SUBAPPLICATION Uebung_006a4 (* SR und T-Flip-Flop mit 3x IE und LinksRechts Baustein *)
  (* Standard: 61499-2; Description: Copyright (c) 2023 Meisterschulen am Ostbahnhof This program and the accompanying materials are made available under the terms of the Eclipse Public License 2.0 which is available at https://www.eclipse.org/legal/epl-2.0/ SPDX-License-Identifier: EPL-2.0 *)
  (* Version 1.0, 2023-10-23, Franz Höpfinger, Meisterschulen am Ostbahnhof *)
  PACKAGE Uebungen;
  IMPORT logiBUS::io::DI::logiBUS_DI::Input_I1;
  IMPORT logiBUS::io::DI::logiBUS_DI::Input_I2;
  IMPORT logiBUS::io::DI::logiBUS_DI::Input_I3;
  IMPORT logiBUS::io::DI::logiBUS_DI_Events::BUTTON_SINGLE_CLICK;
  IMPORT logiBUS::io::DQ::logiBUS_DO::Output_Q1;
  IMPORT logiBUS::io::DQ::logiBUS_DO::Output_Q2;
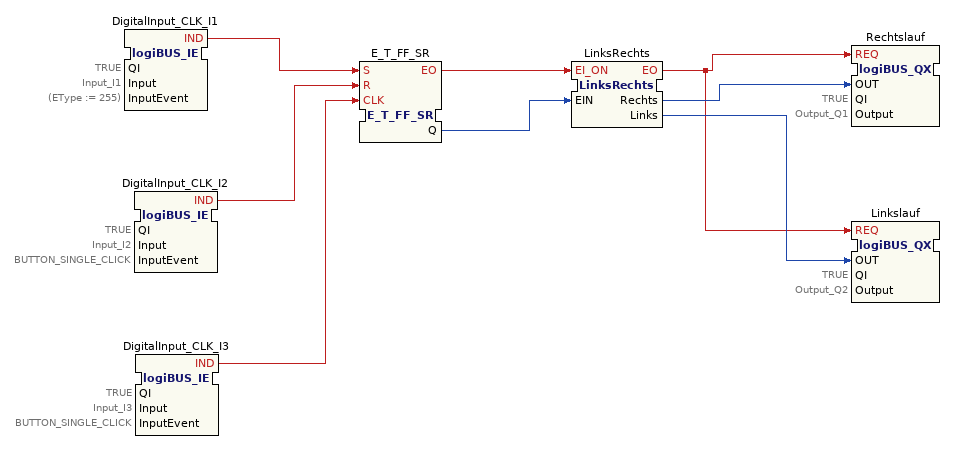
  FBS
    DigitalInput_CLK_I1 : logiBUS::io::DI::logiBUS_IE(QI := TRUE, Input := Input_I1, InputEvent := (EType := 255));
    DigitalInput_CLK_I2 : logiBUS::io::DI::logiBUS_IE(QI := TRUE, Input := Input_I2, InputEvent := BUTTON_SINGLE_CLICK);
    E_T_FF_SR : iec61499::events::E_T_FF_SR;
    DigitalInput_CLK_I3 : logiBUS::io::DI::logiBUS_IE(QI := TRUE, Input := Input_I3, InputEvent := BUTTON_SINGLE_CLICK);
    Rechtslauf : logiBUS::io::DQ::logiBUS_QX(QI := TRUE, Output := Output_Q1);
    Linkslauf : logiBUS::io::DQ::logiBUS_QX(QI := TRUE, Output := Output_Q2);
    LinksRechts : logiBUS::utils::sequence::verteiler::LinksRechts;
  END_FBS
  EVENT_CONNECTIONS
    DigitalInput_CLK_I1.IND TO E_T_FF_SR.S;
    DigitalInput_CLK_I2.IND TO E_T_FF_SR.R;
    DigitalInput_CLK_I3.IND TO E_T_FF_SR.CLK;
    E_T_FF_SR.EO TO LinksRechts.EI_ON;
    LinksRechts.EO TO Linkslauf.REQ;
    LinksRechts.EO TO Rechtslauf.REQ;
  END_CONNECTIONS
  DATA_CONNECTIONS
    LinksRechts.Rechts TO Rechtslauf.OUT;
    E_T_FF_SR.Q TO LinksRechts.EIN;
    LinksRechts.Links TO Linkslauf.OUT;
  END_CONNECTIONS
END_SUBAPPLICATION
